FUNCTION_BLOCK Gate
  (* Standard: 61499-2 *)
  (* Version 0.1, 2017-00-23, hpea485, UOA *)
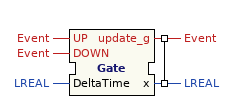
  EVENT_INPUT
    UP;
    DOWN;
  END_EVENT
  EVENT_OUTPUT
    update_g WITH x;
  END_EVENT
  VAR_INPUT
    DeltaTime : LREAL := 0.01;
  END_VAR
  VAR_OUTPUT
    x : LREAL;
  END_VAR
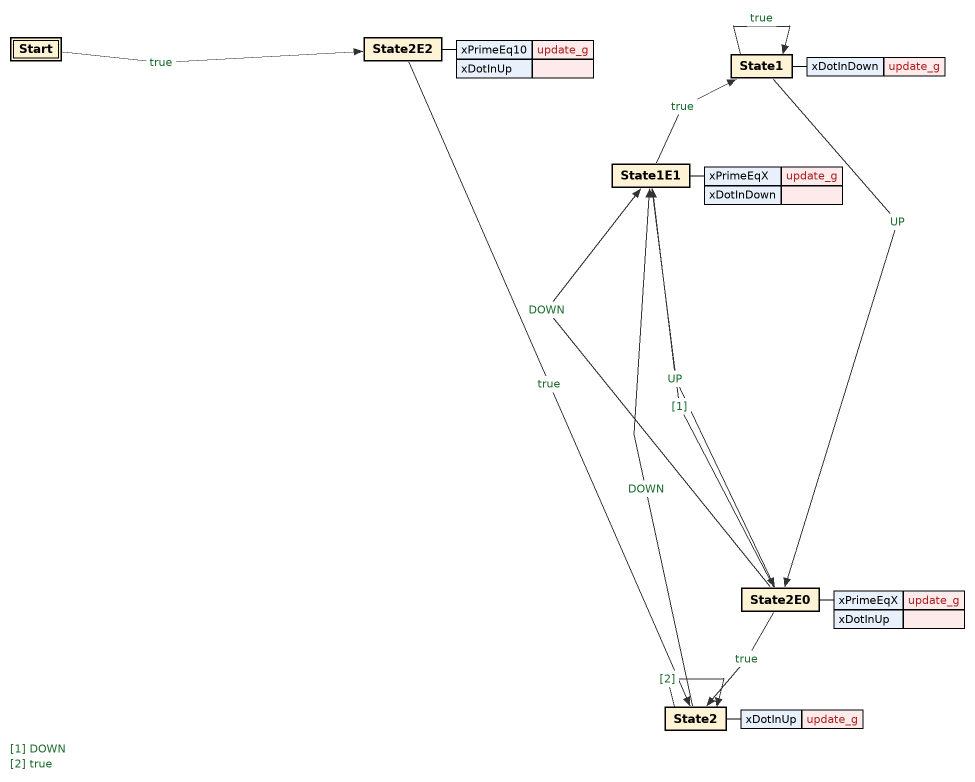
  EC_STATES
    Start;
    State2E2 : xPrimeEq10 -> update_g, xDotInUp;
    State1 : xDotInDown -> update_g;
    State2E0 : xPrimeEqX -> update_g, xDotInUp;
    State2 : xDotInUp -> update_g;
    State1E1 : xPrimeEqX -> update_g, xDotInDown;
  END_STATES
  EC_TRANSITIONS
    Start TO State2E2 := true;
    State2E2 TO State2 := true;
    State2E0 TO State1E1 := DOWN;
    State1 TO State2E0 := UP;
    State1 TO State1 := true;
    State2E0 TO State2 := true;
    State2E0 TO State1E1 := DOWN;
    State2 TO State1E1 := DOWN;
    State2 TO State2 := true;
    State1E1 TO State1 := true;
    State1E1 TO State2E0 := UP;
  END_TRANSITIONS
  ALGORITHM xPrimeEqX IN C: (* ODE_init *)
x_prime = x;
  END_ALGORITHM
  ALGORITHM xPrimeEq10 IN C: (* ODE_init *)
x_prime = 10;
  END_ALGORITHM
  ALGORITHM xDotInDown IN C: (* ODE *)
x_dot = (1 - x) / 2;
  END_ALGORITHM
  ALGORITHM xDotInUp IN C: (* ODE *)
x_dot = (10 - x) / 2;
  END_ALGORITHM
END_FUNCTION_BLOCK
